INTERFACE I_Objekt_Roboter

METHOD M_Reset : BOOL
VAR_INPUT
END_VAR
END_METHOD

METHOD M_Start : BOOL
VAR_INPUT
END_VAR
END_METHOD

METHOD M_Stop : BOOL
VAR_INPUT
END_VAR
END_METHOD

PROPERTY P_Prozessparameter : sRoboterProzessVariablen
SET
END_SET
END_PROPERTY

PROPERTY P_State : eObjectAktorState
GET
END_GET
END_PROPERTY

PROPERTY Test_Param : sRoboterProzessVariablen
GET
END_GET
END_PROPERTY

END_INTERFACE

(* stored: Version 1.1.0.1
   Itf I_Objekt_Roboter: Id {8b7da271-a67b-4341-9ae9-95bafa302d51}
   Method M_Reset: Id {2245070b-0cc0-4022-9bef-6b6ce503cc8c}
   Method M_Start: Id {089b0ebb-61c6-4392-86ed-0651d20f913f}
   Method M_Stop: Id {62f9137f-86dc-4b9e-8ee6-11dfb4ae5fb2}
   Property P_Prozessparameter: Id {108e5dc2-fcea-485f-b838-63c6f5f51ba6}
   Set Set: Id {94154204-fc41-45f9-826f-5377845f788c}
   Property P_State: Id {ea621a6c-f313-43a3-9a01-9581043d7e55}
   Get Get: Id {aa61956f-e124-4b0d-8039-0892f041c089}
   Property Test_Param: Id {9aa13e12-84f5-4f04-8693-ab62001ced60}
   Get Get: Id {635cf7a6-3b6b-4234-bea1-e83af7957871} *)
